INTERFACE ITF_TopElement1 EXTENDS ITF_BaseTopElement

END_INTERFACE

(* stored: Version 1.1.0.1
   Itf ITF_TopElement1: Id {cdc7c8ec-3c0a-02cc-1531-bed4e1783d28} *)
